// Empty function block with no fields, properties, methods, inheritance or interfaces.
FUNCTION_BLOCK FB_Empty
VAR
END_VAR

END_FUNCTION_BLOCK

(* stored: Version 1.1.0.1, ProductVersion 3.1.4024.15
   POU FB_Empty: Id {7d8707a8-603f-4771-ac23-b2c0b5451025}, SpecialFunc None *)
